PROGRAM prgComEffIO
VAR
	fbCom					: FB_MqttCommunicator_V2;
	stringArray_Last_HB		: ARRAY[0..50] OF STRING(30);
END_VAR

fbCom(
	bConnect:= TRUE, 
	strAuthKey:=  'BE736352867778' ,
	sUserName:= 'bd8cddef-7a46-4cb7-9100-c3c67f8ed94a', 
	sUserPassword:= '26bcb4df-2135-49e0-bf55-9c706b8073f9', 
	eSavePositionCertificate:= eSavePositionOnPLC.ePostionHardDisk, 
	bConnected=> , 
	bError=> , 
	hrErrorCode=> , 
	eConnectionState=> , 
	eErrorMessage_Out=> );

END_PROGRAM

(* stored: Version 1.1.0.1, ProductVersion 3.1.4024.12
   POU prgComEffIO: Id {cbcd318b-bf51-484c-bcaa-d6efcdf43fe3}, SpecialFunc None *)
